FUNCTION_BLOCK FB_Test2
VAR_INPUT
		i: INT;
END_VAR
VAR_OUTPUT
END_VAR
VAR

END_VAR

END_FUNCTION_BLOCK

(* stored: Version 1.1.0.1, ProductVersion 3.1.4024.12
   POU FB_Test2: Id {b386e113-997f-4246-baf7-74a116b1bd17}, SpecialFunc None *)
